(* CODESYS project position_control.project

Project tree, tasks and I/O mapping:
  DRV1 : Digitax M750, Nidec Control Techniques, version 1.10.1.9
    application Application
      Task Configuration
        Freewheeling
      program Freewheeling [ST]
    RTEthernet
    Ethernet : Ethernet, Nidec Control Techniques, version 1.10.1.9
    <Empty>
    <Empty>
  DRV2 : Digitax M750, Nidec Control Techniques, version 1.10.1.9
    application Application
      Task Configuration
        Freewheeling
      program Freewheeling [ST]
    RTEthernet
    Ethernet : Ethernet, Nidec Control Techniques, version 1.10.1.9
    MCi210 : MCi210, Nidec Control Techniques, version 1.10.1.9
      application Application
        task Freewheeling (freewheeling, priority 1) calls Freewheeling
        task Position (cyclic, interval t#4ms, priority 6) calls Position
        program Freewheeling [ST]
        program Position [ST]: COUNTER
        global variables GVL
        global variables GVL_1
      RTEthernet
      Ethernet_1 : Ethernet, Nidec Control Techniques, version 1.10.1.9
      PLCopen General Axis Pool
    <Empty>
  Advanced Link Editor
    Section
*)

// DRV2/MCi210/Application/GVL
{attribute 'qualified_only'}
VAR_GLOBAL
END_VAR

// DRV2/MCi210/Application/GVL_1
{attribute 'qualified_only'}
VAR_GLOBAL PERSISTENT RETAIN
END_VAR

// DRV1/Application/Freewheeling
PROGRAM Freewheeling
VAR
END_VAR

END_PROGRAM

// DRV2/Application/Freewheeling
PROGRAM Freewheeling
VAR
END_VAR

END_PROGRAM

// DRV2/MCi210/Application/Freewheeling
PROGRAM Freewheeling
VAR
	Init: BOOL := 0;
	CAM_PARAMETERS: ARRAY[0..9] OF DINT;
END_VAR
VAR RETAIN
	VALUE: INT :=50;
END_VAR

IF Init = 0 THEN
WriteUserParameterBOOL(1,1,19,TRUE);      // Save parameters on power down enable
WriteUserParameterBOOL(1,06,02,TRUE);     // Use high precision speed reference (1.06.01)
Init := 1;

(*CAM_PARAMETERS[0] := 31001;
CAM_PARAMETERS[1] := 32001;
CAM_PARAMETERS[2] := 41001;
CAM_PARAMETERS[3] := 38003;
CAM_PARAMETERS[4] := 39011;
CAM_PARAMETERS[5] := 39009;
*)
M31.P001 := 1;						      // amc enable
M32.P001 := 0;  						  // Select master as SPEED position
M41.P001 := 1;							  // amc enable
M38.P003 := 1092.00*2;					
M39.P011 := 2000;
M39.P009 := 1092.00*2;

CAM_PARAMETERS[6] := 34007;
M34.P007 := 0;

M18.P001 := 1;
END_IF

END_PROGRAM

// DRV2/MCi210/Application/Position
{attribute 'PerformanceCache'}
PROGRAM Position
VAR
	motion_start: BOOL;
	old_motion_start: BOOL;
	PPR: DINT;
	mesafe: DINT;
	pozok: DINT;
	Virtual_speed: DINT;
	output_state: BOOL;
	Home_button: BOOL;
	OldHomeButton: BOOL;
	Homing: BOOL;
	Home_OK : BOOL;
	Home_State: BOOL;
	AMC_MODE_STATE: STRING;
	
		TARGET: DINT;
	COUNT_UP: DINT;
	COUNT_DOWN: DINT;
	TASK_TIME_MSC: DINT;
END_VAR
VAR_OUTPUT
	OUT: LREAL;
	OUT_TEMP: DINT;
END_VAR

PPR := 65536;
motion_start := M18.P031;

pozok:= M33.P004;
output_state:= m08.P005;

Home_button := M18.P042;
//AmcHomingSystem.AmcHomeComplete := M08.P005;
Home_State := M18.P040;

TARGET := M20.P022;
OUT := M33.P005;

COUNT_UP:=1;
COUNT_DOWN :=1;

IF TARGET > OUT THEN 
	OUT_TEMP := OUT_TEMP + (COUNT_UP*TASK_TIME_MSC/1000);
	
	IF OUT_TEMP > TARGET THEN 
		OUT_TEMP := TARGET;
	END_IF
ELSIF TARGET < OUT THEN
	
OUT_TEMP := OUT_TEMP - (COUNT_DOWN*TASK_TIME_MSC/1000);
 
	IF OUT_TEMP < TARGET THEN
		OUT_TEMP := TARGET;
	END_IF
	END_IF
OUT := OUT_TEMP;

 OUT_TEMP := M20.P021;
 M32.P008 := OUT_TEMP;


IF M31.P001 = 0 THEN M31.P001 := 1; END_IF
IF M41.P001 = 0 THEN M41.P001 := 1; END_IF

IF motion_start AND NOT old_motion_start
	THEN
	Home_State := FALSE;
	M18.P031 := 0;
	M34.P007 := 1;		// Reference Select = EGB
	M34.P009 :=1;

	mesafe := M34.P003;	
	output_state := TRUE;
	M06.P030 :=1;
	END_IF
	old_motion_start := motion_Start;
	
		IF pozok = mesafe THEN
			M31.P001 := 0;		// Reference Select = 0
			M34.P009 :=0;
		END_IF
		
		IF output_state AND Home_Button AND NOT OldHomeButton THEN
			AMCReferenceSelector.AmcReferenceSelect := 1;
			AMCHomingSystem.AmcHomeMode := 4;
			m06.P032 := 1;
			Home_OK := TRUE;
			Homing := FALSE;
			
		END_IF
		OldHomeButton := Home_button;
		M18.P031 := 1;
		
		
		IF Home_OK AND NOT Homing THEN
			AMCReferenceSelector.AmcReferenceSelect := 4;
		END_IF
		
		IF AMCReferenceSelector.AmcReferenceSelect = 0 THEN
			AMC_MODE_STATE := 'STOP';
		ELSIF AMCReferenceSelector.AmcReferenceSelect = 1 THEN
			AMC_MODE_STATE := 'POSITION ABS';
		ELSIF AMCReferenceSelector.AmcReferenceSelect = 2 THEN
			AMC_MODE_STATE := 'POSITION ABS';
		ELSIF AMCReferenceSelector.AmcReferenceSelect = 3 THEN
			AMC_MODE_STATE := 'CAM';
		ELSIF AMCReferenceSelector.AmcReferenceSelect = 4 THEN
			AMC_MODE_STATE := 'EGB';
		ELSIF AMCReferenceSelector.AmcReferenceSelect = 5 THEN
			AMC_MODE_STATE := 'HOME';
		ELSIF AMCReferenceSelector.AmcReferenceSelect = 6 THEN
			AMC_MODE_STATE := 'POSITION RELEATIVE';
		ELSE
			AMC_MODE_STATE := 'POSITION PROFILE';
		END_IF
		
		//SYNCHRONIZATION
		
		Position.COUNTER.Counter1.CU := 10;

METHOD COUNTER : CTU
VAR_INPUT
	Counter1: CTU;
	Anlik_deger: WORD :=0;
END_VAR
Counter1.PV := 100;

Counter1(
	CU :=  ,
	RESET :=  ,
	//PV := ,
	Q => ,
	CV => );
	
	Anlik_deger := Counter1;
END_METHOD

END_PROGRAM
